INTERFACE I_NodeExecuteEndEvent EXTENDS I_Event

PROPERTY PUBLIC TargetNode : I_Node
GET
END_GET
END_PROPERTY

END_INTERFACE

(* stored: Version 1.1.0.1, ProductVersion 3.1.4024.12
   Itf I_NodeExecuteEndEvent: Id {dc59c47f-79c1-06cd-1d36-bf0bace27a27}
   Property TargetNode: Id {5f04d79d-9843-046b-0dad-dfb25789b913}
   Get Get: Id {c5344353-93be-0b9f-3ec5-017e603210b7} *)
